FUNCTION_BLOCK MeasurementBuffer
VAR
	MemRingBuffer : FB_MemRingBuffer;
	BufferArray : ARRAY[0..GVL.MAX_BUFFER_SIZE] OF BYTE;
	
END_VAR

METHOD AddMeasurement
VAR_INPUT
END_VAR
END_METHOD

END_FUNCTION_BLOCK

(* stored: Version 1.1.0.1, ProductVersion 3.1.4024.12
   POU MeasurementBuffer: Id {1650884d-214c-4b9b-a209-9988b5b3841b}, SpecialFunc None
   Method AddMeasurement: Id {e38050eb-d64a-4f20-af81-a387013f37cc} *)
